KUKA KRL program: chk_w2_wechs_ok.src

&ACCESS RVO3
&REL 1
&COMMENT GUN C1
DEF chk_w2_wechs_ok( )

; VERIFICAÇÃO DE FERRAMENTA: C1

$TIMER[10] = 0
$TIMER_STOP[10] = FALSE

wait for (($IN[585]) and ($IN[577]) and ($in[161]) and (($in[177]) or (NOT ($in[177]) and $in[3320])) and ($in[193]) and (not $in[209]) and ($IN[201]) and ($in[169]) and ($in[185]) AND ($in[219]))

$TIMER_STOP[10] = TRUE
$TIMER[10] = 0

;//---- End -------
;Diag_Appl(#Off,5)
END
